DATA_BLOCK "dbArchiveControlEom"
{ S7_Optimized_Access := 'TRUE' }
VERSION : 0.8
NON_RETAIN
"fbArchiveControlEom"

BEGIN

END_DATA_BLOCK

